FUNCTION_BLOCK ABSTRACT FBA_LinearDrive_1 IMPLEMENTS I_LinearDrive
VAR_INPUT
	bEnable : BOOL;
	sensorDefaultState : BOOL;
END_VAR
VAR_OUTPUT	
	ready : BOOL;
END_VAR
VAR
	direction : MC_Direction;
	
	step : Homing;
	homingComplete : BOOL;
	
	home AT %I* : BOOL;
END_VAR

PROPERTY ABSTRACT Active : BOOL
GET
END_GET
END_PROPERTY

{attribute 'monitoring':='call'}
PROPERTY AtHome : BOOL
GET
AtHome := home <> sensorDefaultState;
END_GET
END_PROPERTY

PROPERTY ABSTRACT Error : BOOL
GET
END_GET
END_PROPERTY

{attribute 'monitoring':='call'}
PROPERTY HomeSet : BOOL
GET
HomeSet := homingComplete;
END_GET
END_PROPERTY

METHOD ABSTRACT homingSequence : BOOL
VAR_INPUT
END_VAR
END_METHOD

METHOD ABSTRACT reset : BOOL
VAR_INPUT
END_VAR
END_METHOD

METHOD ABSTRACT stop : BOOL
VAR_INPUT
END_VAR
END_METHOD

METHOD ABSTRACT toHome : BOOL
VAR_INPUT
END_VAR
END_METHOD

END_FUNCTION_BLOCK

(* stored: Version 1.1.0.1, ProductVersion 3.1.4024.11
   POU FBA_LinearDrive_1: Id {3e72b5a2-ae17-4fe1-887a-049c7204ae1e}, SpecialFunc None
   Folder Abstract: Id {099c3586-f9c4-45ef-91a4-939c2346bbf4}
   Folder Properties: Id {34d59db6-d915-44ee-8f75-ab2b60266802}
   Property Active: Id {b4345cfa-7780-4342-af00-8b0c9dd31a39}
   Get Get: Id {e5995cc4-91ec-4f3f-b94e-36aea69719da}
   Property AtHome: Id {1e5c0658-e3c1-4c64-be47-7ee92f06252f}
   Get Get: Id {6ed66d09-10f2-43cb-9edc-6276afa0c3b7}
   Property Error: Id {a250a152-a560-4a57-9725-1b8a8a8d9a88}
   Get Get: Id {3a8bb637-e694-4202-97c1-05f27af11d02}
   Property HomeSet: Id {a3e1cf87-7de6-45b5-ae06-358dcc38e4ea}
   Get Get: Id {b875dea1-716c-4fe0-a42d-353eaf9023fc}
   Method homingSequence: Id {4ae133e7-1755-4dcf-93bb-b5fb2152291f}
   Method reset: Id {7b7ecfe5-7494-4566-8ea2-0a6bbf68b261}
   Method stop: Id {9547cd59-8c39-428e-b5ec-69995e192197}
   Method toHome: Id {efb4e337-16c9-41d9-9b22-ac92fc8868d3} *)
